// TIA Portal V16 export
// export: Created 2021-11-12T13:31:12.8855146Z, ExportSetting WithDefaults, DisplayName Totally Integrated Automation Portal, DisplayVersion V16 Update 3, DisplayName TIA Portal Version Control Interface, DisplayVersion V16 Update 2, DisplayName TIA Portal Openness, DisplayVersion V16 Update 3, DisplayName SINAMICS Startdrive Advanced, DisplayVersion V16 Update 5, DisplayName SINAMICS Startdrive G130, G150, S120, S150, SINAMICS MV, S210, DisplayVersion V16 Update 5, DisplayName SINAMICS Startdrive G110M, G120, G120C, G120D, G120P, G115D, DisplayVersion V16 Update 5, DisplayName STEP 7 Professional, DisplayVersion V16 Update 3, DisplayName STEP 7 Safety, DisplayVersion V16, DisplayName WinCC UA Professional, DisplayVersion V16 Update 3
DATA_BLOCK "Sfty_Comm"   // DB4, F_DB
{ S7_Optimized_Access := 'TRUE'; DB_Accessible_From_OPC_UA := 'FALSE' }
VERSION : 0.1
// stored: AutoNumber true, DBAccessibleFromOPCUA false
   VAR
      Inputs : Bool;
      BSN1_2_in { S7_SetPoint := 'True'} : "UDT_COMM_F_BSN1_2_CRS";   // Safety inputs from owen BSN1 a BSN2
      BSN1_2_out { S7_SetPoint := 'True'} : "UDT_COMM_F_CRS_BSN1_2";   // Safety outputs to owen BSN1 a BSN2
      BSN3_in { S7_SetPoint := 'True'} : "UDT_COMM_F_BSN3_CRS";   // Safety inputs from owen BSN3
      BSN3_out { S7_SetPoint := 'True'} : "UDT_COMM_F_CRS_BSN3";   // Safety outputs to owen BSN3
      BSN4_5_in { S7_SetPoint := 'True'} : "UDT_COMM_F_BSN4_5_CRS";   // Safety inputs from owen BSN4 a 5
      BSN4_5_out { S7_SetPoint := 'True'} : "UDT_COMM_F_CRS_BSN4_5";   // Safety outputs to owen BSN4 a 5
      SCH1_in { S7_SetPoint := 'True'} : "UDT_COMM_F_SCH1_CRS";   // Safety inputs from press SCH1
      SCH1_out { S7_SetPoint := 'True'} : "UDT_COMM_F_CRS_SCH1";   // Safety outputs to press SCH1
      "1R1+RC01_In" { S7_SetPoint := 'True'} : "UDT_DriveRobotABB_ControllerSftyDI";   // Safety inputs from robot controller 1R1+RC01
      "1R1+RC01_Out" { S7_SetPoint := 'True'} : "UDT_DriveRobotABB_ControllerSftyDO";   // Safety outputs fom robot controller 1R1+RC01
      "1R2+RC01_In" { S7_SetPoint := 'True'} : "UDT_DriveRobotABB_ControllerSftyDI";   // Safety inputs from robot controller 1R2+RC01
      "1R2+RC01_Out" { S7_SetPoint := 'True'} : "UDT_DriveRobotABB_ControllerSftyDO";   // Safety outputs fom robot controller 1R2+RC01
      "1R3_4+RC01_In" { S7_SetPoint := 'True'} : "UDT_DriveRobotABB_ControllerSftyDI";   // Safety inputs from robot controller 1R3+RC01
      "1R3_4+RC01_Out" { S7_SetPoint := 'True'} : "UDT_DriveRobotABB_ControllerSftyR3_4_DO";   // Safety outputs fom robot controller 1R3+RC01
      "1R5+RC01_In" { S7_SetPoint := 'True'} : "UDT_DriveRobotABB_ControllerSftyDI";   // Safety inputs from robot controller 1R5+RC01
      "1R5+RC01_Out" { S7_SetPoint := 'True'} : "UDT_DriveRobotABB_ControllerSftyDO";   // Safety outputs fom robot controller 1R5+RC01
      "1R6+RC01_In" { S7_SetPoint := 'True'} : "UDT_DriveRobotABB_ControllerSftyDI";   // Safety inputs from robot controller 1R6+RC01
      "1R6+RC01_Out" { S7_SetPoint := 'True'} : "UDT_DriveRobotABB_ControllerSftyDO";   // Safety outputs fom robot controller 1R6+RC01
      "2R1+RC01_In" { S7_SetPoint := 'True'} : "UDT_DriveRobotABB_ControllerSftyDI";   // Safety inputs from robot controller 2R1+RC01
      "2R1+RC01_Out" { S7_SetPoint := 'True'} : "UDT_DriveRobotABB_ControllerSftyDO";   // Safety outputs fom robot controller 2R1+RC01
      "2R2+RC01_In" { S7_SetPoint := 'True'} : "UDT_DriveRobotABB_ControllerSftyDI";   // Safety inputs from robot controller 2R2+RC01
      "2R2+RC01_Out" { S7_SetPoint := 'True'} : "UDT_DriveRobotABB_ControllerSftyDO";   // Safety outputs fom robot controller 2R2+RC01
      "110+UC12-TA01_F_In" { S7_SetPoint := 'True'} : "UDT_CU240E_I_30";   // Safety inputs inverter 110+UC12-TA01
      "120+UC12-TA01_F_In" { S7_SetPoint := 'True'} : "UDT_CU240E_I_30";   // Safety inputs inverter 120+UC12-TA01
      "210+UC12-TA01_F_In" { S7_SetPoint := 'True'} : "UDT_CU240E_I_30";   // Safety inputs inverter 210+UC12-TA01
      "220+UC12-TA01_F_In" { S7_SetPoint := 'True'} : "UDT_CU240E_I_30";   // Safety inputs inverter 220+UC12-TA01
      "230+UC12-TA01_F_In" { S7_SetPoint := 'True'} : "UDT_CU240E_I_30";   // Safety inputs inverter 230+UC12-TA01
      "230+UC12-TA02_F_In" { S7_SetPoint := 'True'} : "UDT_CU240E_I_30";   // Safety inputs inverter 230+UC12-TA02
      "320+UC21-TA01_F_In" { S7_SetPoint := 'True'} : "UDT_CU240E_I_30";   // Safety inputs inverter 320+UC21-TA01
      "330+UC21-TA01_F_In" { S7_SetPoint := 'True'} : "UDT_CU240E_I_30";   // Safety inputs inverter 330+UC21-TA01
      "330+UC21-TA02_F_In" { S7_SetPoint := 'True'} : "UDT_CU240E_I_30";   // Safety inputs inverter 330+UC21-TA02
      "330+UC21-TA03_F_In" { S7_SetPoint := 'True'} : "UDT_CU240E_I_30";   // Safety inputs inverter 330+UC21-TA03
      "430+UC21-TA01_F_In" { S7_SetPoint := 'True'} : "UDT_CU240E_I_30";   // Safety inputs inverter 430+UC21-TA01
      "440+UC21-TA01_F_In" { S7_SetPoint := 'True'} : "UDT_CU240E_I_30";   // Safety inputs inverter 440+UC21-TA01
      "450+UC21-TA01_F_In" { S7_SetPoint := 'True'} : "UDT_CU240E_I_30";   // Safety inputs inverter 450+UC21-TA01
      "450+UC21-TA02_F_In" { S7_SetPoint := 'True'} : "UDT_CU240E_I_30";   // Safety inputs inverter 450+UC21-TA02
      "450+UC21-TA03_F_In" { S7_SetPoint := 'True'} : "UDT_CU240E_I_30";   // Safety inputs inverter 450+UC21-TA03
      "450+UC21-TA04_F_In" { S7_SetPoint := 'True'} : "UDT_CU240E_I_30";   // Safety inputs inverter 450+UC21-TA04
      "460+UC21-TA01_F_In" { S7_SetPoint := 'True'} : "UDT_CU240E_I_30";   // Safety inputs inverter 460+UC21-TA01
      "460+UC21-TA02_F_In" { S7_SetPoint := 'True'} : "UDT_CU240E_I_30";   // Safety inputs inverter 460+UC21-TA02
      "460+UC21-TA03_F_In" { S7_SetPoint := 'True'} : "UDT_CU240E_I_30";   // Safety inputs inverter 460+UC21-TA03
      "460+UC21-TA04_F_In" { S7_SetPoint := 'True'} : "UDT_CU240E_I_30";   // Safety inputs inverter 460+UC21-TA04
      "110+UC12-TA01_F_Out" { S7_SetPoint := 'True'} : "UDT_CU240E_O_30";   // Safety outputs inverter 110+UC12-TA01
      "120+UC12-TA01_F_Out" { S7_SetPoint := 'True'} : "UDT_CU240E_O_30";   // Safety outputs inverter 120+UC12-TA01
      "210+UC12-TA01_F_Out" { S7_SetPoint := 'True'} : "UDT_CU240E_O_30";   // Safety outputs inverter 210+UC12-TA01
      "220+UC12-TA01_F_Out" { S7_SetPoint := 'True'} : "UDT_CU240E_O_30";   // Safety outputs inverter 220+UC12-TA01
      "230+UC12-TA01_F_Out" { S7_SetPoint := 'True'} : "UDT_CU240E_O_30";   // Safety outputs inverter 230+UC12-TA01
      "230+UC12-TA02_F_Out" { S7_SetPoint := 'True'} : "UDT_CU240E_O_30";   // Safety outputs inverter 230+UC12-TA02
      "320+UC21-TA01_F_Out" { S7_SetPoint := 'True'} : "UDT_CU240E_O_30";   // Safety outputs inverter 320+UC21-TA01
      "330+UC21-TA01_F_Out" { S7_SetPoint := 'True'} : "UDT_CU240E_O_30";   // Safety outputs inverter 330+UC21-TA01
      "330+UC21-TA02_F_Out" { S7_SetPoint := 'True'} : "UDT_CU240E_O_30";   // Safety outputs inverter 330+UC21-TA02
      "330+UC21-TA03_F_Out" { S7_SetPoint := 'True'} : "UDT_CU240E_O_30";   // Safety outputs inverter 330+UC21-TA03
      "430+UC21-TA01_F_Out" { S7_SetPoint := 'True'} : "UDT_CU240E_O_30";   // Safety outputs inverter 430+UC21-TA01
      "440+UC21-TA01_F_Out" { S7_SetPoint := 'True'} : "UDT_CU240E_O_30";   // Safety outputs inverter 440+UC21-TA01
      "450+UC21-TA01_F_Out" { S7_SetPoint := 'True'} : "UDT_CU240E_O_30";   // Safety outputs inverter 450+UC21-TA01
      "450+UC21-TA02_F_Out" { S7_SetPoint := 'True'} : "UDT_CU240E_O_30";   // Safety outputs inverter 450+UC21-TA02
      "450+UC21-TA03_F_Out" { S7_SetPoint := 'True'} : "UDT_CU240E_O_30";   // Safety outputs inverter 450+UC21-TA03
      "450+UC21-TA04_F_Out" { S7_SetPoint := 'True'} : "UDT_CU240E_O_30";   // Safety outputs inverter 450+UC21-TA04
      "460+UC21-TA01_F_Out" { S7_SetPoint := 'True'} : "UDT_CU240E_O_30";   // Safety outputs inverter 460+UC21-TA01
      "460+UC21-TA02_F_Out" { S7_SetPoint := 'True'} : "UDT_CU240E_O_30";   // Safety outputs inverter 460+UC21-TA02
      "460+UC21-TA03_F_Out" { S7_SetPoint := 'True'} : "UDT_CU240E_O_30";   // Safety outputs inverter 460+UC21-TA03
      "460+UC21-TA04_F_Out" { S7_SetPoint := 'True'} : "UDT_CU240E_O_30";   // Safety outputs inverter 460+UC21-TA04
   END_VAR
BEGIN
END_DATA_BLOCK
